ABB RobotStudio station: Asignación2_1.rsstn

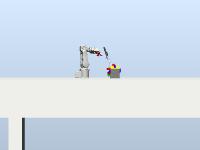
Station Asignación2 (saved by RobotStudio 6.8.8307.1040)
Controller System1, task T_ROB1: task frame (RAPID world) sits at (0, 0, 4135) mm in the station
Controller System1
  mechanical unit ROB_1: IRB120_3_58__01_2, 6 joints, base frame (0, 0, 0) mm
Layout (positions relative to the parent item):
  - FlexPendant [part, from Equipment\FlexPendant.rslib] at (-1461.15, 1249.2, 744.39) mm
  - IRC5_Control-Module [part, from Equipment\IRC5_Control-Module.rslib] at (-1307.51, 1231.51, 100) mm, rotated rx 90 ry 0 rz 90 deg
  - IRB120_3_58__01_2 [mechanism, from Robots\IRB120_3_58_G_01.rslib] at (0, 0, 4135) mm; joint values [0.3641, -0.1044, 0.2488, -0.5086, 0.6141, 0.658] (rad or m)
  - Binzel_air_22_2 [mechanism, from Tools\Binzel_air_22.rslib] at (319.13, 100, 4675.02) mm, rotated rx 180 ry 52 rz 180 deg
  - Part_4 [part] at (0, 0, 4135) mm
  - Table mod1_3 [part] at (-10400, -11700, 0) mm
Attachment: Binzel_air_22_2 is attached to IRB120_3_58__01_2 / Link6
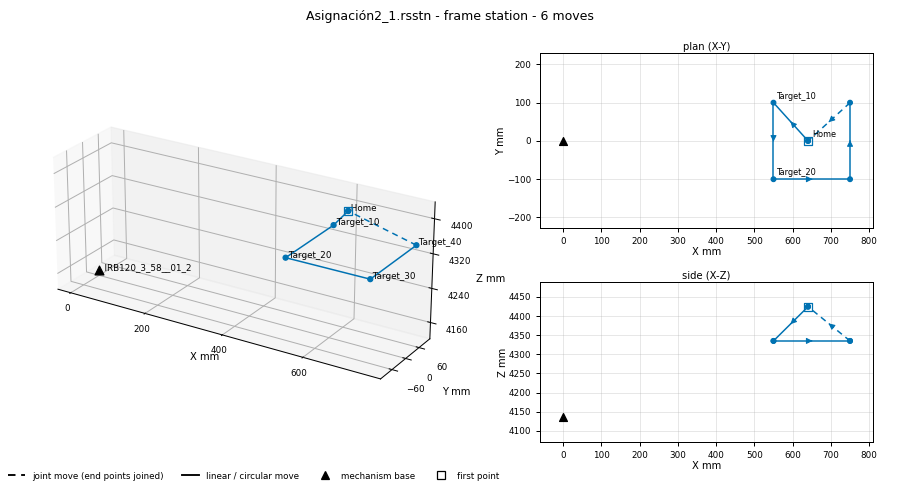
[picture p0: tool path of Asignación2_1.rsstn in frame station, 6 of 6 moves have a stored position in this frame; points joined in program order, loops and branches not executed]
Targets, tools, work objects and paths stored in the station, written as RAPID:
! task T_ROB1
MODULE CalibData
  PERS tooldata tWeldGun:=[TRUE,[[125.800591275,0,391.268161315],[0.898794046,0,0.438371147,0]],[3,[0,0,100],[0,1,0,0],0,0,0]];
  TASK PERS wobjdata Workobject_1:=[FALSE,TRUE,"",[[0,0,0],[1,0,0,0]],[[500.1655,49.8345,100],[0.820028671,-0.42556594,0.176275184,-0.339666997]]];
ENDMODULE

! task T_ROB1
MODULE Module1
  CONST robtarget Home:=[[640.301700826,0,289.419411487],[0.069756473,0,0.99756405,0],[0,0,0,0],[9E+09,9E+09,9E+09,9E+09,9E+09,9E+09]];
  CONST robtarget Target_10:=[[-0.234052335,-41.066234567,115.384419999],[0.176275184,-0.339666997,0.820028671,0.42556594],[0,0,0,0],[9E+09,9E+09,9E+09,9E+09,9E+09,9E+09]];
  CONST robtarget Target_20:=[[141.187303884,-122.474219299,-0.256143936],[0.176275184,-0.339666997,0.820028671,0.42556594],[0,0,0,0],[9E+09,9E+09,9E+09,9E+09,9E+09,9E+09]];
  CONST robtarget Target_30:=[[282.608660139,-41.066234588,115.384419969],[0.176275184,-0.339666997,0.820028671,0.42556594],[0,0,0,0],[9E+09,9E+09,9E+09,9E+09,9E+09,9E+09]];
  CONST robtarget Target_40:=[[141.18730392,40.341750143,231.024983903],[0.176275184,-0.339666997,0.820028671,0.42556594],[0,0,0,0],[9E+09,9E+09,9E+09,9E+09,9E+09,9E+09]];
  PROC Path_10()
    MoveJ Home,v300,fine,tWeldGun\WObj:=wobj0;
    MoveL Target_10,v300,fine,tWeldGun\WObj:=Workobject_1;
    MoveL Target_20,v300,fine,tWeldGun\WObj:=Workobject_1;
    MoveL Target_30,v300,fine,tWeldGun\WObj:=Workobject_1;
    MoveL Target_40,v300,fine,tWeldGun\WObj:=Workobject_1;
    MoveJ Home,v300,fine,tWeldGun\WObj:=wobj0;
  ENDPROC
ENDMODULE

